// TIA Portal project "UR_PLC_MODBUS_TEST" (V15.1)
// Este es un programa de prueba para comunicar un PLC a un contenedor de Docker que ejecuta una estación robótica virtual a través del protocolo MODBUS TCP/IP

(* hardware
DEVICE "S7-1200 station_1"  S7-1200 Station
   slot 0: "Rack_0"  S7-1200 Rack  Rack  V1.0
   slot 1: "PLC_1"  CPU 1215C AC/DC/Rly  6ES7 215-1BG40-0XB0  V4.2
*)

// ===== PLC "PLC_1"  CPU 1215C AC/DC/Rly =====

VAR_GLOBAL   // PLC tag table "Tabla de variables estándar"
   "btn_1_redundant" AT %M0.0 : Bool;
   "btn_1" AT %I0.0 : Bool;
   "Tag_1" AT %Q0.0 : Bool;
   "Tag_2" AT %Q0.1 : Bool;
   "Tag_3" AT %M0.2 : Bool;
   "Clock_Byte" AT %MB200 : Byte;
   "Clock_10Hz" AT %M200.0 : Bool;
   "Clock_5Hz" AT %M200.1 : Bool;
   "Clock_2.5Hz" AT %M200.2 : Bool;
   "Clock_2Hz" AT %M200.3 : Bool;
   "Clock_1.25Hz" AT %M200.4 : Bool;
   "Clock_1Hz" AT %M200.5 : Bool;
   "Clock_0.625Hz" AT %M200.6 : Bool;
   "Clock_0.5Hz" AT %M200.7 : Bool;
END_VAR

DATA_BLOCK "DATOS_Client"   // DB2
{ S7_Optimized_Access := 'TRUE' }
VERSION : 0.1
   VAR
      DISCONNECT : Bool;
      MODE : USInt := 1;   // Modo 1: Modo de escritura
      DATA_ADDR : UDInt := 40129;   // 4XXXX: Direcciones de escritura en registros de retención remoto
      DATA_LEN : UInt := 1;   // Longitud: 16 bits = 1 palabra = 1 registro
      CONNECT : TCON_IP_v4;
      DONE : Bool;
      BUSY : Bool;
      ERROR : Bool;
      STATUS : Word;
      BUFFER : Word := 16#1;
   END_VAR
BEGIN
   CONNECT.InterfaceId := 64;
   CONNECT.ID := 1;
   CONNECT.ConnectionType := 11;
   CONNECT.RemoteAddress.ADDR[1] := 192;
   CONNECT.RemoteAddress.ADDR[2] := 168;
   CONNECT.RemoteAddress.ADDR[3] := 105;
   CONNECT.RemoteAddress.ADDR[4] := 32;
   CONNECT.RemotePort := 502;
   CONNECT.ActiveEstablished := true;
   CONNECT.LocalPort := 0;
END_DATA_BLOCK

DATA_BLOCK "DATOS_Server"   // DB4
{ S7_Optimized_Access := 'TRUE' }
VERSION : 0.1
   VAR
      DISCONNECT : Bool;
      MB_HOLD_REG : Word;
      CONNECT : TCON_IP_v4;
      NDR : Bool;
      DR : Bool;
      ERROR : Bool;
      STATUS : Word;
   END_VAR
BEGIN
END_DATA_BLOCK

ORGANIZATION_BLOCK "Main"   // OB1, LAD, ProgramCycle
TITLE = "Main Program Sweep (Cycle)"
{ S7_Optimized_Access := 'TRUE' }
VERSION : 0.1
   VAR_INPUT
      Initial_Call : Bool;   // Initial call of this OB
      Remanence : Bool;   // =True, if remanent data are available
   END_VAR
BEGIN

REGION Network 1
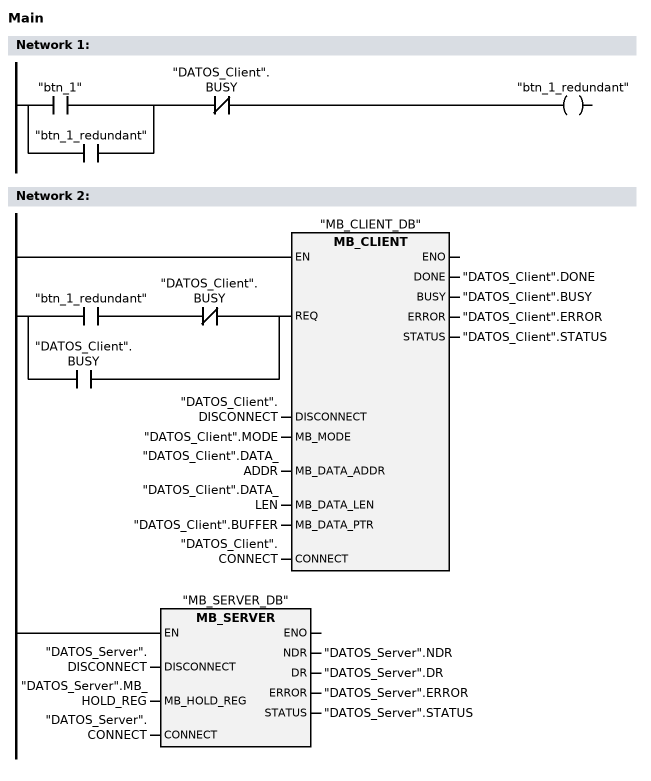
   RUNG wire#powerrail
      Contact( "btn_1" )
      wire#w1
      I_Contact( "DATOS_Client".BUSY )
      Coil( "btn_1_redundant" )
   END_RUNG
   RUNG wire#powerrail
      Contact( "btn_1_redundant" )
   END_RUNG wire#w1
   // the same network as SCL:
   "btn_1_redundant" := ("btn_1" OR "btn_1_redundant") AND NOT "DATOS_Client".BUSY;
END_REGION

REGION Network 2
   "MB_CLIENT_DB"(REQ := ("btn_1_redundant" AND NOT "DATOS_Client".BUSY) OR "DATOS_Client".BUSY,   // MB_CLIENT
                  DISCONNECT := "DATOS_Client".DISCONNECT,
                  MB_MODE := "DATOS_Client".MODE,
                  MB_DATA_ADDR := "DATOS_Client".DATA_ADDR,
                  MB_DATA_LEN := "DATOS_Client".DATA_LEN,
                  MB_DATA_PTR := "DATOS_Client".BUFFER,
                  CONNECT := "DATOS_Client".CONNECT,
                  DONE => "DATOS_Client".DONE,
                  BUSY => "DATOS_Client".BUSY,
                  ERROR => "DATOS_Client".ERROR,
                  STATUS => "DATOS_Client".STATUS);
   "MB_SERVER_DB"(DISCONNECT := "DATOS_Server".DISCONNECT,   // MB_SERVER
                  MB_HOLD_REG := "DATOS_Server".MB_HOLD_REG,
                  CONNECT := "DATOS_Server".CONNECT,
                  NDR => "DATOS_Server".NDR,
                  DR => "DATOS_Server".DR,
                  ERROR => "DATOS_Server".ERROR,
                  STATUS => "DATOS_Server".STATUS);
END_REGION
END_ORGANIZATION_BLOCK